FUNCTION_BLOCK T_LidApplyStation EXTENDS T_Station
VAR_INPUT
END_VAR
VAR_OUTPUT
END_VAR
VAR
	processState : (IDLE,EXTEND_APPLICATOR_ARM, WAIT,RETRACT_APPLICATOR_ARM, COMPLETE);
	waitTimer : TON;
	cylinder : I_Cylinder; 
END_VAR
VAR CONSTANT
	PROCESS_TIME : TIME := T#2S;
END_VAR

super^();

METHOD PROTECTED Execute
VAR_INPUT
END_VAR


CASE processState OF
	
	IDLE : // 
	
		waitTimer(IN:=FALSE);
		processState := EXTEND_APPLICATOR_ARM;
	
	EXTEND_APPLICATOR_ARM : // 
	
		cylinder.Extend();
		processState := WAIT;
	
	WAIT : //
	
		waitTimer(IN:=TRUE, PT:=PROCESS_TIME);
		IF waitTimer.Q THEN
			processState := RETRACT_APPLICATOR_ARM;
		END_IF
	
	RETRACT_APPLICATOR_ARM : //
	
		cylinder.Retract();
		processState := COMPLETE;
	
	COMPLETE: //
	
		StateComplete();
		processState := IDLE;

END_CASE
END_METHOD

METHOD FB_init : BOOL
VAR_INPUT
	bInitRetains : BOOL; // if TRUE, the retain variables are initialized (warm start / cold start)
	bInCopyCode : BOOL;  // if TRUE, the instance afterwards gets moved into the copy code (online change)
	Cylinder : I_Cylinder;
END_VAR
this^.cylinder := Cylinder;
END_METHOD

END_FUNCTION_BLOCK

(* stored: Version 1.1.0.1, ProductVersion 3.1.4024.4
   POU T_LidApplyStation: Id {ba5b0c5d-a171-41ee-a5ea-366ebc327b95}, SpecialFunc None
   Method Execute: Id {4a41d72c-d121-41a4-9221-b45ba23d7293}
   Method FB_init: Id {5ce9571e-dbf5-4aa5-939d-cb6f8741dc0a} *)
